FUNCTION TryConvert_ULINT_TO_LREAL : BOOL
VAR_INPUT
	in : ULINT;
	out : REFERENCE TO LREAL;
END_VAR

out := ULINT_TO_LREAL(in);
TryConvert_ULINT_TO_LREAL := TRUE;

END_FUNCTION

(* stored: Version 1.1.0.1, ProductVersion 3.1.4024.12
   POU TryConvert_ULINT_TO_LREAL: Id {7cc647d1-dfa5-4f4a-90de-b5a8717ccf69}, SpecialFunc None *)
